Staubli VAL3: session_change.pgx

program session_change(string x_sName (dimensions=1), bool& x_bResult (dimensions=1))
  local num i
  local string l_sEmpty
  local string l_sEvent
begin
  // check if exist
  // clean the string
  l_sEmpty=""
  x_bResult=false
  if cycleStatus:bCycle==false and cycleStatus:bSimulation==false
    // search inside the sSession
    for i=0 to size(sSessionList)-1
      if x_sName==sSessionList[i]
        // the session exist
        call saveData:changeSession(x_sName)
        // reload the processList
        call processList:loadProcessList(i)
        if i!=0
          popUpMsg("error loading: "+toString("",i))
        else
          // the session has been changed
          x_bResult=true
        endIf
        //
        if !x_bResult
          // not found
          popUpMsg("session not FOUND....")
        endIf
        // reset the homing trajectory
        cycleStatus:bHomeLoaded=false
        // refresh
        use:bUseRefresh=true
        return
      endIf
    endFor
  endIf
  //
end
